// TwinCAT 3 PLC project ConveyorPLC
// ProgramVersion: 3.1.4026.24
// libraries:
//   Tc2_Standard, * (Beckhoff Automation GmbH)
//   Tc2_System, * (Beckhoff Automation GmbH)
// project tree:
//   DUTs/ E_MachineState.TcDUT, ST_ConveyorStatus.TcDUT
//   FBs/ FB_Conveyor.TcPOU
//   GVLs/ GVL_HMI_Operator.TcGVL
//   / PlcTask.TcTTO
//   POUs/ MAIN.TcPOU
// real-time tasks:
//   TASK PlcTask: cycle T#10ms, priority 20, ADS port 350

CONFIGURATION ConveyorPLC
    RESOURCE PLC ON TwinCAT3
        TASK PlcTask(INTERVAL := T#10ms, PRIORITY := 20);
        PROGRAM MAIN WITH PlcTask : MAIN;
    END_RESOURCE
END_CONFIGURATION

// ---- DUTs/E_MachineState.TcDUT
TYPE E_MachineState :
(
    Stopped := 0,
    Starting := 10,
    Running := 20,
    Stopping := 30,
    Faulted := 100
);
END_TYPE

// ---- DUTs/ST_ConveyorStatus.TcDUT
TYPE ST_ConveyorStatus :
STRUCT
    eState          : E_MachineState;

    bMotorRunning   : BOOL;

    bEntrySensor    : BOOL;
    bExitSensor     : BOOL;

    bFaultActive    : BOOL;

    nPartCount      : UDINT;
END_STRUCT
END_TYPE

// ---- GVLs/GVL_HMI_Operator.TcGVL
{attribute 'qualified_only'}
VAR_GLOBAL

    //==============================
    // Operator Commands
    //==============================

    bStartCommand      : BOOL := FALSE;
    bStopCommand       : BOOL := FALSE;
    bResetCommand      : BOOL := FALSE;
    bEmergencyStop     : BOOL := FALSE;

    //==============================
    // Status shown on the HMI
    //==============================

    stStatus           : ST_ConveyorStatus;

END_VAR

// ---- POUs/MAIN.TcPOU
PROGRAM MAIN
VAR
    fbConveyor : FB_Conveyor;
END_VAR

fbConveyor(
    bStart         := GVL_HMI_Operator.bStartCommand,
    bStop          := GVL_HMI_Operator.bStopCommand,
    bReset         := GVL_HMI_Operator.bResetCommand,
    bEmergencyStop := GVL_HMI_Operator.bEmergencyStop
);

GVL_HMI_Operator.stStatus := fbConveyor.stStatus;

END_PROGRAM

// ---- FBs/FB_Conveyor.TcPOU
FUNCTION_BLOCK FB_Conveyor

VAR_INPUT
    bStart          : BOOL;
    bStop           : BOOL;
    bReset          : BOOL;
    bEmergencyStop  : BOOL;
END_VAR

VAR_OUTPUT
    stStatus        : ST_ConveyorStatus;
END_VAR

VAR
    rStart : R_TRIG;
    rStop  : R_TRIG;
    rReset : R_TRIG;
END_VAR

rStart(CLK := bStart);
rStop(CLK := bStop);
rReset(CLK := bReset);

// Emergency Stop has the highest priority
IF bEmergencyStop THEN
    stStatus.eState := E_MachineState.Faulted;
END_IF;

// Reset clears the fault
IF rReset.Q THEN
    stStatus.eState := E_MachineState.Stopped;
END_IF;

// Main machine state
CASE stStatus.eState OF

    E_MachineState.Stopped:

        stStatus.bMotorRunning := FALSE;

        IF rStart.Q THEN
            stStatus.eState := E_MachineState.Starting;
        END_IF


    E_MachineState.Starting:

        stStatus.bMotorRunning := TRUE;
        stStatus.eState := E_MachineState.Running;


    E_MachineState.Running:

        stStatus.bMotorRunning := TRUE;

        IF rStop.Q THEN
            stStatus.eState := E_MachineState.Stopping;
        END_IF


    E_MachineState.Stopping:

        stStatus.bMotorRunning := FALSE;
        stStatus.eState := E_MachineState.Stopped;


    E_MachineState.Faulted:

        stStatus.bMotorRunning := FALSE;

END_CASE;

END_FUNCTION_BLOCK
